(* IEC 61131-3 sources: pandora/pandora/aws-platform-main/aws-platform-main/test/Mocks/Utils/Heartbeat, 1 file *)

(* ---- HeartbeatMock.st ---- *)
USING Esab.Mock;

NAMESPACE Esab.Utils.Heartbeat.Mock

    CLASS HeartbeatMock IMPLEMENTS IHeartbeat
        VAR PUBLIC
            ExecuteMock : MethodMock;
            AliveMock : BoolMethodMock;
            DeadMock : BoolMethodMock;
        END_VAR

        METHOD PUBLIC MockReset
            ExecuteMock.Reset();
            AliveMock.Reset();
            DeadMock.Reset();
        END_METHOD

        METHOD PUBLIC Execute
            ExecuteMock.IncrementCallCount();
        END_METHOD

        METHOD PUBLIC Alive : BOOL
            AliveMock.IncrementCallCount();
            Alive := AliveMock.Value;
        END_METHOD

        METHOD PUBLIC Dead : BOOL
            DeadMock.IncrementCallCount();
            Dead := DeadMock.Value;
        END_METHOD
    END_CLASS

END_NAMESPACE
